% RSLogix 500 project CONVEYER_BAK003.RSS, saved by version 8.30.00.16 %
PROJECT "UNTITLED"    % processor: Bul.1763 MicroLogix 1100 Series B %

PROGRAM FILES
  LAD 2   6 rungs

DATA FILES
  O0 OUTPUT  4 elements
  I1 INPUT  6 elements
  S2 STATUS  66 elements
  B3 BINARY  1 elements
  T4 TIMER  2 elements
  C5 COUNTER  1 elements
  R6 CONTROL  1 elements
  N7 INTEGER  1 elements
  F8 FLOAT  1 elements

LADDER 2
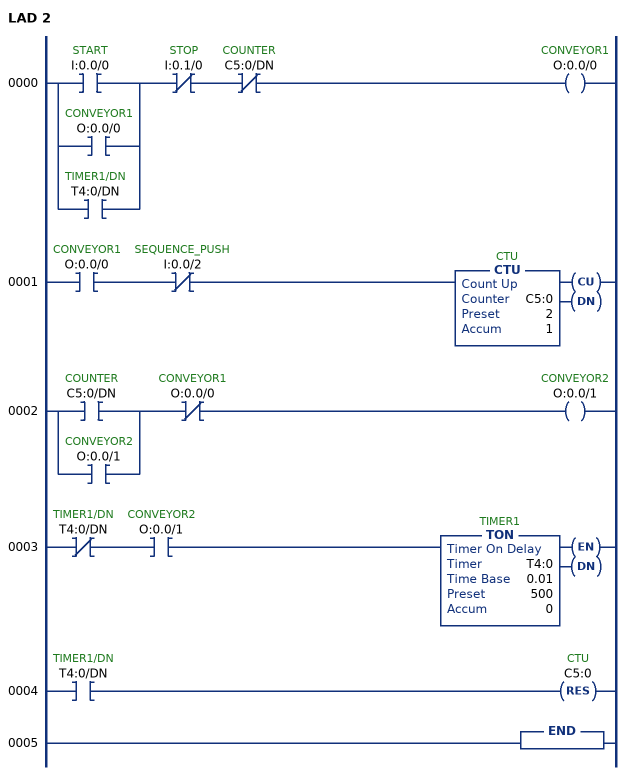
% Rung: 0 %
SOR BST XIC I:0.0/0 NXB BST XIC O:0.0/0 NXB XIC T4:0/DN BND BND XIO I:0.1/0 XIO C5:0/DN OTE O:0.0/0 EOR
%   I:0.0/0  START %
%   O:0.0/0  CONVEYOR1 %
%   T4:0  TIMER1 %
%   I:0.1/0  STOP %
%   C5:0/DN  COUNTER %
% Rung: 1 %
SOR XIC O:0.0/0 XIO I:0.0/2 CTU C5:0 2 1 EOR
%   O:0.0/0  CONVEYOR1 %
%   I:0.0/2  SEQUENCE_PUSH %
%   C5:0  CTU %
% Rung: 2 %
SOR BST XIC C5:0/DN NXB XIC O:0.0/1 BND XIO O:0.0/0 OTE O:0.0/1 EOR
%   C5:0/DN  COUNTER %
%   O:0.0/1  CONVEYOR2 %
%   O:0.0/0  CONVEYOR1 %
% Rung: 3 %
SOR XIO T4:0/DN XIC O:0.0/1 TON T4:0 0.01 500 0 EOR
%   T4:0  TIMER1 %
%   O:0.0/1  CONVEYOR2 %
% Rung: 4 %
SOR XIC T4:0/DN RES C5:0 EOR
%   T4:0  TIMER1 %
%   C5:0  CTU %
% Rung: 5 %
SOR END EOR

OTHER DOCUMENTED ADDRESSES
  T4:1  SEQUENCE_TIMER

DATA TABLE (non-zero values as saved)
DATA T4
% .PRE .ACC %
% T4:0 % 500 0
% T4:1 % 500 116
DATA C5
% .PRE .ACC %
% C5:0 % 2 1
